{attribute addProperty BoxType "KL2641-0001"}
{attribute addProperty Id "Channel_1Channel_DB7D35B100"}
{attribute addProperty CRC "240938105"}
{attribute addProperty SizeInBites "0"}
{attribute addProperty SizeInBytes "0"}
TYPE KL_0E5C6C79 :
STRUCT
	{attribute addProperty Name "Channel_1"}
	Channel_1 : Channel_DB7D35B1;
END_STRUCT
END_TYPE

(* stored: Version 1.2.0.0, ProductVersion 3.1.4024.9
   DUT KL_0E5C6C79: Id {dc0031c5-4c33-4989-86df-7f5f7617514d} *)
